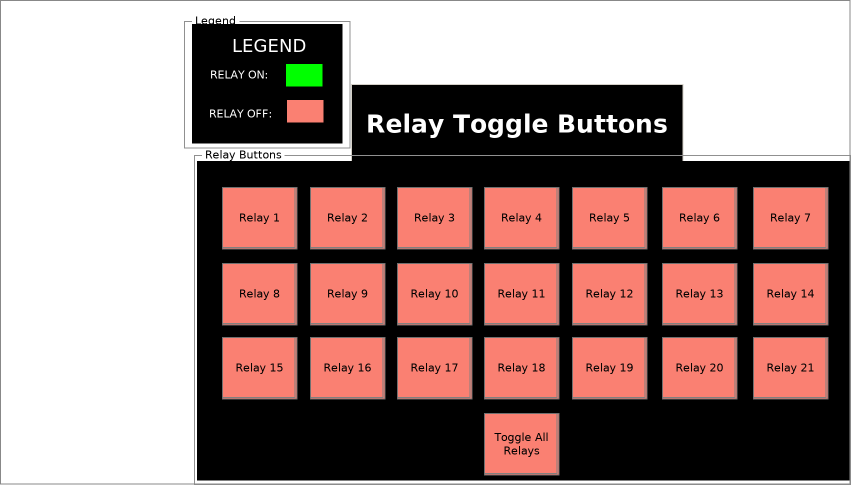
VISUALIZATION Visualization  // 851x485
    Textfield (351,84 332x79), "Relay Toggle Buttons"
    GroupBox (194,147 657x338), "Relay Buttons"
        Rectangle (3,14 653x319)
        Button (28,40 75x62), "Relay 1", colour toggle: BoolRelayArray[1]
            toggle BoolRelayArray[1]
        Button (116,40 75x62), "Relay 2", colour toggle: BoolRelayArray[2]
            toggle BoolRelayArray[2]
        Button (203,40 75x62), "Relay 3", colour toggle: BoolRelayArray[3]
            toggle BoolRelayArray[3]
        Button (290,40 75x62), "Relay 4", colour toggle: BoolRelayArray[4]
            toggle BoolRelayArray[4]
        Button (28,116 75x62), "Relay 8", colour toggle: BoolRelayArray[8]
            toggle BoolRelayArray[8]
        Button (116,116 75x62), "Relay 9", colour toggle: BoolRelayArray[9]
            toggle BoolRelayArray[9]
        Button (116,190 75x62), "Relay 16", colour toggle: BoolRelayArray[16]
            toggle BoolRelayArray[16]
        Button (203,190 75x62), "Relay 17", colour toggle: BoolRelayArray[17]
            toggle BoolRelayArray[17]
        Button (203,116 75x62), "Relay 10", colour toggle: BoolRelayArray[10]
            toggle BoolRelayArray[10]
        Button (290,190 75x62), "Relay 18", colour toggle: BoolRelayArray[18]
            toggle BoolRelayArray[18]
        Button (378,190 75x62), "Relay 19", colour toggle: BoolRelayArray[19]
            toggle BoolRelayArray[19]
        Button (468,190 75x62), "Relay 20", colour toggle: BoolRelayArray[20]
            toggle BoolRelayArray[20]
        Button (559,190 75x62), "Relay 21", colour toggle: BoolRelayArray[21]
            toggle BoolRelayArray[21]
        Button (290,116 75x62), "Relay 11", colour toggle: BoolRelayArray[11]
            toggle BoolRelayArray[11]
        Button (378,116 75x62), "Relay 12", colour toggle: BoolRelayArray[12]
            toggle BoolRelayArray[12]
        Button (468,116 75x62), "Relay 13", colour toggle: BoolRelayArray[13]
            toggle BoolRelayArray[13]
        Button (559,116 75x62), "Relay 14", colour toggle: BoolRelayArray[14]
            toggle BoolRelayArray[14]
        Button (559,40 75x62), "Relay 7", colour toggle: BoolRelayArray[7]
            toggle BoolRelayArray[7]
        Button (468,40 75x62), "Relay 6", colour toggle: BoolRelayArray[6]
            toggle BoolRelayArray[6]
        Button (378,40 75x62), "Relay 5", colour toggle: BoolRelayArray[5]
            toggle BoolRelayArray[5]
        Button (28,190 75x62), "Relay 15", colour toggle: BoolRelayArray[15]
            toggle BoolRelayArray[15]
        Button (290,266 75x62), "Toggle All Relays", colour toggle: MAIN.ToggleAllRelaysButton
            toggle MAIN.ToggleAllRelaysButton
    Rectangle (197,161 653x319)
    Button (222,187 75x62), "Relay 1", colour toggle: BoolRelayArray[1]
        toggle BoolRelayArray[1]
    Button (310,187 75x62), "Relay 2", colour toggle: BoolRelayArray[2]
        toggle BoolRelayArray[2]
    Button (397,187 75x62), "Relay 3", colour toggle: BoolRelayArray[3]
        toggle BoolRelayArray[3]
    Button (484,187 75x62), "Relay 4", colour toggle: BoolRelayArray[4]
        toggle BoolRelayArray[4]
    Button (222,263 75x62), "Relay 8", colour toggle: BoolRelayArray[8]
        toggle BoolRelayArray[8]
    Button (310,263 75x62), "Relay 9", colour toggle: BoolRelayArray[9]
        toggle BoolRelayArray[9]
    Button (310,337 75x62), "Relay 16", colour toggle: BoolRelayArray[16]
        toggle BoolRelayArray[16]
    Button (397,337 75x62), "Relay 17", colour toggle: BoolRelayArray[17]
        toggle BoolRelayArray[17]
    Button (397,263 75x62), "Relay 10", colour toggle: BoolRelayArray[10]
        toggle BoolRelayArray[10]
    Button (484,337 75x62), "Relay 18", colour toggle: BoolRelayArray[18]
        toggle BoolRelayArray[18]
    Button (572,337 75x62), "Relay 19", colour toggle: BoolRelayArray[19]
        toggle BoolRelayArray[19]
    Button (662,337 75x62), "Relay 20", colour toggle: BoolRelayArray[20]
        toggle BoolRelayArray[20]
    Button (753,337 75x62), "Relay 21", colour toggle: BoolRelayArray[21]
        toggle BoolRelayArray[21]
    Button (484,263 75x62), "Relay 11", colour toggle: BoolRelayArray[11]
        toggle BoolRelayArray[11]
    Button (572,263 75x62), "Relay 12", colour toggle: BoolRelayArray[12]
        toggle BoolRelayArray[12]
    Button (662,263 75x62), "Relay 13", colour toggle: BoolRelayArray[13]
        toggle BoolRelayArray[13]
    Button (753,263 75x62), "Relay 14", colour toggle: BoolRelayArray[14]
        toggle BoolRelayArray[14]
    Button (753,187 75x62), "Relay 7", colour toggle: BoolRelayArray[7]
        toggle BoolRelayArray[7]
    Button (662,187 75x62), "Relay 6", colour toggle: BoolRelayArray[6]
        toggle BoolRelayArray[6]
    Button (572,187 75x62), "Relay 5", colour toggle: BoolRelayArray[5]
        toggle BoolRelayArray[5]
    Button (222,337 75x62), "Relay 15", colour toggle: BoolRelayArray[15]
        toggle BoolRelayArray[15]
    Button (484,413 75x62), "Toggle All Relays", colour toggle: MAIN.ToggleAllRelaysButton
        toggle MAIN.ToggleAllRelaysButton
    GroupBox (184,13 166x135), "Legend"
        Rectangle (8,11 150x119)
        Textfield (34,18 103x30), "LEGEND"
        Textfield (23,47 72x30), "RELAY ON:"
        Textfield (22,86 76x30), "RELAY OFF:"
        Rectangle (101,50 38x24)
        Rectangle (102,86 38x24)
    Rectangle (192,24 150x119)
    Textfield (218,31 103x30), "LEGEND"
    Textfield (207,60 72x30), "RELAY ON:"
    Textfield (206,99 76x30), "RELAY OFF:"
    Rectangle (285,63 38x24)
    Rectangle (286,99 38x24)
END_VISUALIZATION

(* stored: Version 1.1.0.1, ProductVersion 3.1.4024.13
   Visu Visualization: Id {9b059ab3-f918-45c6-b370-6da0cdcdda94} *)
